TYPE ST_Vector3 :
STRUCT
    x : LREAL;
    y : LREAL;
    z : LREAL;
END_STRUCT
END_TYPE

(* stored: Version 1.1.0.1, ProductVersion 3.1.4026.18
   DUT ST_Vector3: Id {cb3d564d-c5ae-45eb-a7d2-908db1297cce} *)
